FUNCTION_BLOCK Automatik
VAR_INPUT
END_VAR
VAR_OUTPUT
END_VAR
VAR
END_VAR

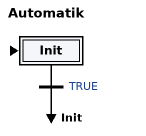
INITIAL_STEP Init:
END_STEP
TRANSITION FROM Init TO Init
    := TRUE;
END_TRANSITION

END_FUNCTION_BLOCK

(* stored: Version 1.1.0.1, ProductVersion 3.1.4024.4
   POU Automatik: Id {65e8707b-8cf8-4c30-8ee7-9ed839cf8731}, SpecialFunc None *)
